PROGRAM F21_ContentHandScanner
VAR
	bDT_HandScanerInUse			: BOOL;
	fbBarcodeType			: FB_SYSTEM_BarcodeType;

	bPackBarcode					: BOOL;
	bOuterIntermediateBarcode		: BOOL;
	bOuterBarcode					: BOOL;
	bCaseBarcode					: BOOL;
	sPackBarcode					: T_PACK_Barcode;
	sOuterIntermediateBarcode		:  T_MaxString;
	sOuterBarcode					: T_OUTER_Barcode;
	sCaseBarcode					: T_CASE_Barcode;

	bLocalCaseBarcode					: BOOL;
	sLocalCaseBarcode					: T_CASE_Barcode;

	fbSearchCaseContent	: FB_SYSTEM_SearchBarcode;

	fbFindOCV_DB			: FB_OCV_FindDB;
	fbFindOAC_DB			: FB_OAC_FindDB;

(*	fbFindOCVFile			: FB_OCV_FindFile;
	stOACData				: ST_OAC_Data;
	sCode				: T_PACK_Barcode;*)

	aOCVRecordDBName		 : ARRAY[1..2] OF T_MaxString;
	sOACRecordName			: T_MaxString;


	fbRestoreCACDataFromDB	:FB_CAC_RestoreDataFromDB;
	sCACFile				: T_MaxString;

	nOCVRestored			: UDINT;
	nOACRestored			: UDINT;
	nCACRestored			: UDINT;

	bOACFound: BOOL;
	bOCVFound: BOOL;
	bOCVValid: BOOL;
	sOuterCodeAI		: T_MaxString;
	(*strPackCodeAI:			STRING(255);*)

	bValidateForOCVDataExistDone :BOOL;
	bValidateForRefeedDone: BOOL;
	bValidateForRefeedOK: BOOL;

	rtrigValidateOCVForDataExistValid			: R_TRIG;
	rtrigValidateOCVForDataExistInvalid			: R_TRIG;
	rtrigValidateOCVForDataNotExist			: R_TRIG;
	tofValidateOCVForDataExisValid			: TOF;
	tofValidateOCVForDataExisInvalid			: TOF;
	tofValidateOCVForDataNotExis				: TOF;


	rtrigValidateOACForRefeedDoneValid		: R_TRIG;
	rtrigValidateOACForRefeedDoneInvalid		: R_TRIG;
	rtrigValidateOACForDataNotExist			: R_TRIG;
	tofValidateOACForRefeedValid			: TOF;
	tofValidateOACForRefeedInvalid			: TOF;
	tofValidateOACForDataNotExis				: TOF;

	rtrigRestoreCACFileDoneValid: R_TRIG;
	rtrigRestoreCACFileDoneInvalid: R_TRIG;
	tofRestoreCACFileValid: TOF;
	tofRestoreCACFileInvalid: TOF;

END_VAR

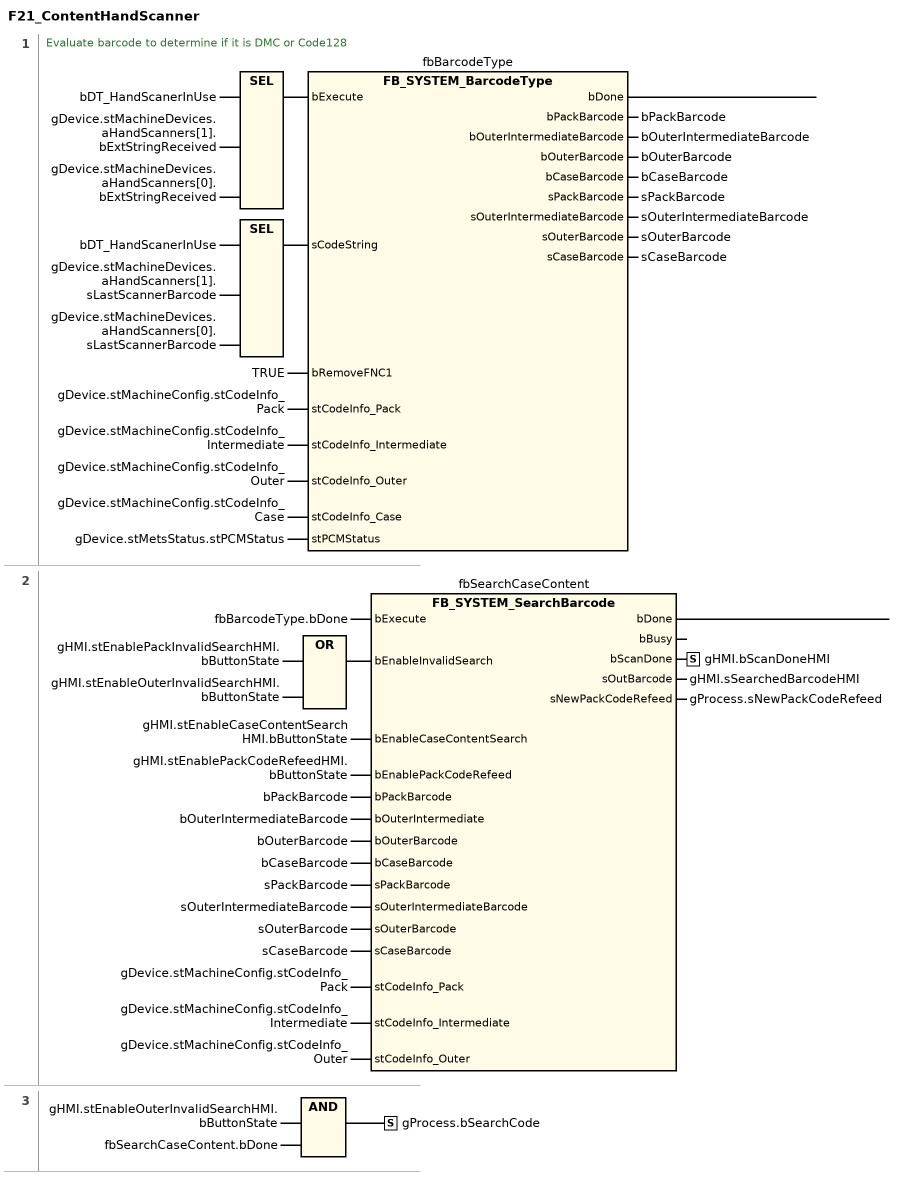
// NETWORK 1
// Evaluate barcode to determine if it is DMC or Code128
fbBarcodeType(
    bExecute := SEL(bDT_HandScanerInUse, gDevice.stMachineDevices.aHandScanners[1].bExtStringReceived, gDevice.stMachineDevices.aHandScanners[0].bExtStringReceived),
    sCodeString := SEL(bDT_HandScanerInUse, gDevice.stMachineDevices.aHandScanners[1].sLastScannerBarcode, gDevice.stMachineDevices.aHandScanners[0].sLastScannerBarcode),
    bRemoveFNC1 := TRUE,
    stCodeInfo_Pack := gDevice.stMachineConfig.stCodeInfo_Pack,
    stCodeInfo_Intermediate := gDevice.stMachineConfig.stCodeInfo_Intermediate,
    stCodeInfo_Outer := gDevice.stMachineConfig.stCodeInfo_Outer,
    stCodeInfo_Case := gDevice.stMachineConfig.stCodeInfo_Case,
    stPCMStatus := gDevice.stMetsStatus.stPCMStatus,
    bPackBarcode => bPackBarcode,
    bOuterIntermediateBarcode => bOuterIntermediateBarcode,
    bOuterBarcode => bOuterBarcode,
    bCaseBarcode => bCaseBarcode,
    sPackBarcode => sPackBarcode,
    sOuterIntermediateBarcode => sOuterIntermediateBarcode,
    sOuterBarcode => sOuterBarcode,
    sCaseBarcode => sCaseBarcode); // FB_SYSTEM_BarcodeType

// NETWORK 2
fbSearchCaseContent(
    bExecute := fbBarcodeType.bDone,
    bEnableInvalidSearch := gHMI.stEnablePackInvalidSearchHMI.bButtonState OR gHMI.stEnableOuterInvalidSearchHMI.bButtonState,
    bEnableCaseContentSearch := gHMI.stEnableCaseContentSearchHMI.bButtonState,
    bEnablePackCodeRefeed := gHMI.stEnablePackCodeRefeedHMI.bButtonState,
    bPackBarcode := bPackBarcode,
    bOuterIntermediate := bOuterIntermediateBarcode,
    bOuterBarcode := bOuterBarcode,
    bCaseBarcode := bCaseBarcode,
    sPackBarcode := sPackBarcode,
    sOuterIntermediateBarcode := sOuterIntermediateBarcode,
    sOuterBarcode := sOuterBarcode,
    sCaseBarcode := sCaseBarcode,
    stCodeInfo_Pack := gDevice.stMachineConfig.stCodeInfo_Pack,
    stCodeInfo_Intermediate := gDevice.stMachineConfig.stCodeInfo_Intermediate,
    stCodeInfo_Outer := gDevice.stMachineConfig.stCodeInfo_Outer,
    sOutBarcode => gHMI.sSearchedBarcodeHMI,
    sNewPackCodeRefeed => gProcess.sNewPackCodeRefeed); // FB_SYSTEM_SearchBarcode
gHMI.bScanDoneHMI S= fbSearchCaseContent.bScanDone;

// NETWORK 3
gProcess.bSearchCode S= gHMI.stEnableOuterInvalidSearchHMI.bButtonState AND fbSearchCaseContent.bDone;

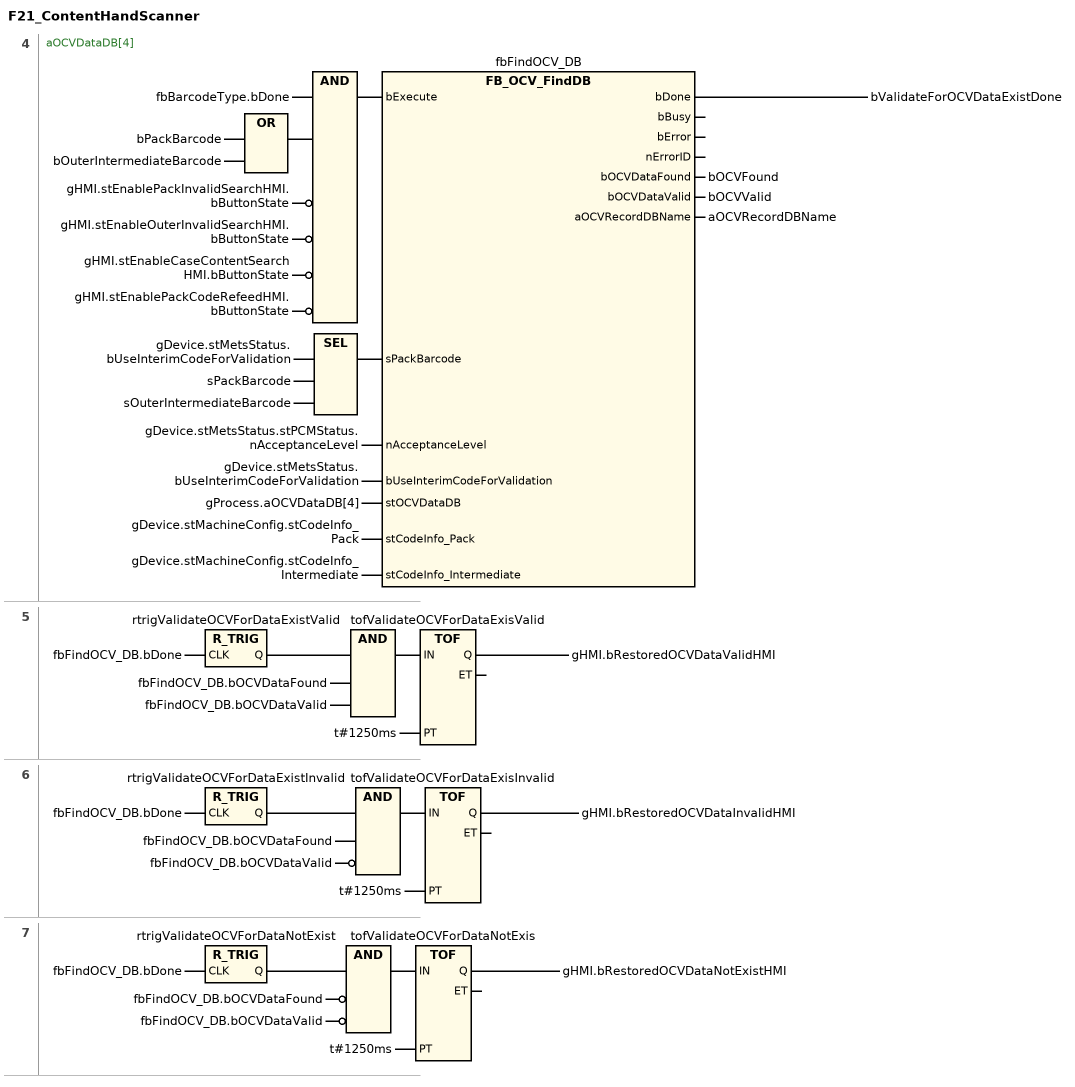
// NETWORK 4
// aOCVDataDB[4]
fbFindOCV_DB(
    bExecute := fbBarcodeType.bDone AND (bPackBarcode OR bOuterIntermediateBarcode) AND NOT gHMI.stEnablePackInvalidSearchHMI.bButtonState AND NOT gHMI.stEnableOuterInvalidSearchHMI.bButtonState AND NOT gHMI.stEnableCaseContentSearchHMI.bButtonState AND NOT gHMI.stEnablePackCodeRefeedHMI.bButtonState,
    sPackBarcode := SEL(gDevice.stMetsStatus.bUseInterimCodeForValidation, sPackBarcode, sOuterIntermediateBarcode),
    nAcceptanceLevel := gDevice.stMetsStatus.stPCMStatus.nAcceptanceLevel,
    bUseInterimCodeForValidation := gDevice.stMetsStatus.bUseInterimCodeForValidation,
    stOCVDataDB := gProcess.aOCVDataDB[4],
    stCodeInfo_Pack := gDevice.stMachineConfig.stCodeInfo_Pack,
    stCodeInfo_Intermediate := gDevice.stMachineConfig.stCodeInfo_Intermediate,
    bOCVDataFound => bOCVFound,
    bOCVDataValid => bOCVValid,
    aOCVRecordDBName => aOCVRecordDBName); // FB_OCV_FindDB
bValidateForOCVDataExistDone := fbFindOCV_DB.bDone;

// NETWORK 5
rtrigValidateOCVForDataExistValid(CLK := fbFindOCV_DB.bDone); // R_TRIG
tofValidateOCVForDataExisValid(IN := rtrigValidateOCVForDataExistValid.Q AND fbFindOCV_DB.bOCVDataFound AND fbFindOCV_DB.bOCVDataValid, PT := t#1250ms); // TOF
gHMI.bRestoredOCVDataValidHMI := tofValidateOCVForDataExisValid.Q;

// NETWORK 6
rtrigValidateOCVForDataExistInvalid(CLK := fbFindOCV_DB.bDone); // R_TRIG
tofValidateOCVForDataExisInvalid(IN := rtrigValidateOCVForDataExistInvalid.Q AND fbFindOCV_DB.bOCVDataFound AND NOT fbFindOCV_DB.bOCVDataValid, PT := t#1250ms); // TOF
gHMI.bRestoredOCVDataInvalidHMI := tofValidateOCVForDataExisInvalid.Q;

// NETWORK 7
rtrigValidateOCVForDataNotExist(CLK := fbFindOCV_DB.bDone); // R_TRIG
tofValidateOCVForDataNotExis(IN := rtrigValidateOCVForDataNotExist.Q AND NOT fbFindOCV_DB.bOCVDataFound AND NOT fbFindOCV_DB.bOCVDataValid, PT := t#1250ms); // TOF
gHMI.bRestoredOCVDataNotExistHMI := tofValidateOCVForDataNotExis.Q;

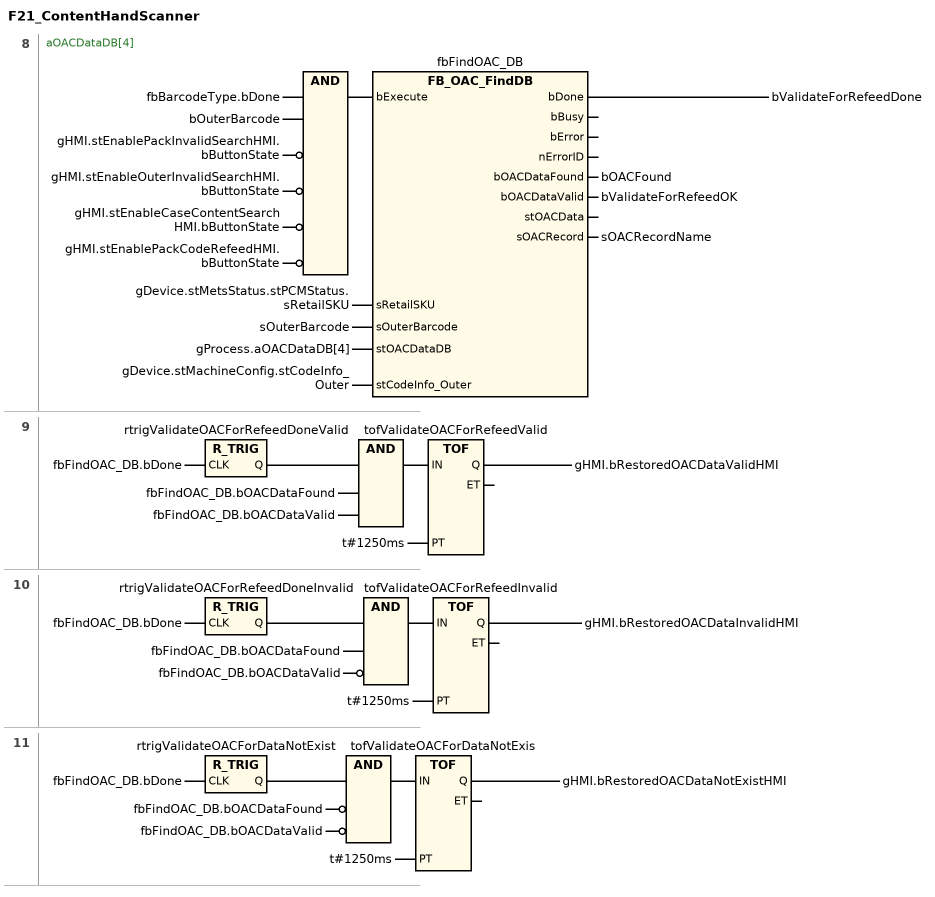
// NETWORK 8
// aOACDataDB[4]
fbFindOAC_DB(
    bExecute := fbBarcodeType.bDone AND bOuterBarcode AND NOT gHMI.stEnablePackInvalidSearchHMI.bButtonState AND NOT gHMI.stEnableOuterInvalidSearchHMI.bButtonState AND NOT gHMI.stEnableCaseContentSearchHMI.bButtonState AND NOT gHMI.stEnablePackCodeRefeedHMI.bButtonState,
    sRetailSKU := gDevice.stMetsStatus.stPCMStatus.sRetailSKU,
    sOuterBarcode := sOuterBarcode,
    stOACDataDB := gProcess.aOACDataDB[4],
    stCodeInfo_Outer := gDevice.stMachineConfig.stCodeInfo_Outer,
    bOACDataFound => bOACFound,
    bOACDataValid => bValidateForRefeedOK,
    sOACRecord => sOACRecordName); // FB_OAC_FindDB
bValidateForRefeedDone := fbFindOAC_DB.bDone;

// NETWORK 9
rtrigValidateOACForRefeedDoneValid(CLK := fbFindOAC_DB.bDone); // R_TRIG
tofValidateOACForRefeedValid(IN := rtrigValidateOACForRefeedDoneValid.Q AND fbFindOAC_DB.bOACDataFound AND fbFindOAC_DB.bOACDataValid, PT := t#1250ms); // TOF
gHMI.bRestoredOACDataValidHMI := tofValidateOACForRefeedValid.Q;

// NETWORK 10
rtrigValidateOACForRefeedDoneInvalid(CLK := fbFindOAC_DB.bDone); // R_TRIG
tofValidateOACForRefeedInvalid(IN := rtrigValidateOACForRefeedDoneInvalid.Q AND fbFindOAC_DB.bOACDataFound AND NOT fbFindOAC_DB.bOACDataValid, PT := t#1250ms); // TOF
gHMI.bRestoredOACDataInvalidHMI := tofValidateOACForRefeedInvalid.Q;

// NETWORK 11
rtrigValidateOACForDataNotExist(CLK := fbFindOAC_DB.bDone); // R_TRIG
tofValidateOACForDataNotExis(IN := rtrigValidateOACForDataNotExist.Q AND NOT fbFindOAC_DB.bOACDataFound AND NOT fbFindOAC_DB.bOACDataValid, PT := t#1250ms); // TOF
gHMI.bRestoredOACDataNotExistHMI := tofValidateOACForDataNotExis.Q;

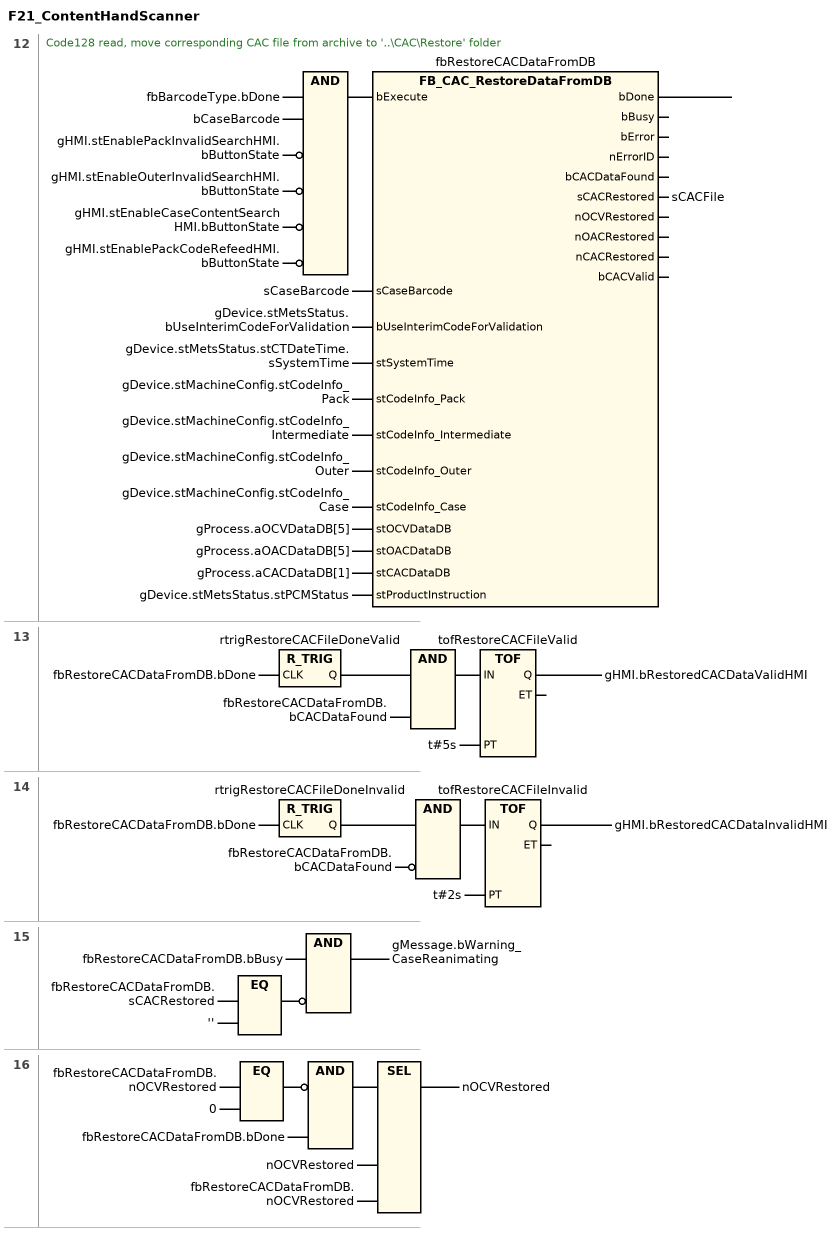
// NETWORK 12
// Code128 read, move corresponding CAC file from archive to '..\CAC\Restore' folder
fbRestoreCACDataFromDB(
    bExecute := fbBarcodeType.bDone AND bCaseBarcode AND NOT gHMI.stEnablePackInvalidSearchHMI.bButtonState AND NOT gHMI.stEnableOuterInvalidSearchHMI.bButtonState AND NOT gHMI.stEnableCaseContentSearchHMI.bButtonState AND NOT gHMI.stEnablePackCodeRefeedHMI.bButtonState,
    sCaseBarcode := sCaseBarcode,
    bUseInterimCodeForValidation := gDevice.stMetsStatus.bUseInterimCodeForValidation,
    stSystemTime := gDevice.stMetsStatus.stCTDateTime.sSystemTime,
    stCodeInfo_Pack := gDevice.stMachineConfig.stCodeInfo_Pack,
    stCodeInfo_Intermediate := gDevice.stMachineConfig.stCodeInfo_Intermediate,
    stCodeInfo_Outer := gDevice.stMachineConfig.stCodeInfo_Outer,
    stCodeInfo_Case := gDevice.stMachineConfig.stCodeInfo_Case,
    stOCVDataDB := gProcess.aOCVDataDB[5],
    stOACDataDB := gProcess.aOACDataDB[5],
    stCACDataDB := gProcess.aCACDataDB[1],
    stProductInstruction := gDevice.stMetsStatus.stPCMStatus,
    sCACRestored => sCACFile); // FB_CAC_RestoreDataFromDB

// NETWORK 13
rtrigRestoreCACFileDoneValid(CLK := fbRestoreCACDataFromDB.bDone); // R_TRIG
tofRestoreCACFileValid(IN := rtrigRestoreCACFileDoneValid.Q AND fbRestoreCACDataFromDB.bCACDataFound, PT := t#5s); // TOF
gHMI.bRestoredCACDataValidHMI := tofRestoreCACFileValid.Q;

// NETWORK 14
rtrigRestoreCACFileDoneInvalid(CLK := fbRestoreCACDataFromDB.bDone); // R_TRIG
tofRestoreCACFileInvalid(IN := rtrigRestoreCACFileDoneInvalid.Q AND NOT fbRestoreCACDataFromDB.bCACDataFound, PT := t#2s); // TOF
gHMI.bRestoredCACDataInvalidHMI := tofRestoreCACFileInvalid.Q;

// NETWORK 15
gMessage.bWarning_CaseReanimating := fbRestoreCACDataFromDB.bBusy AND NOT (fbRestoreCACDataFromDB.sCACRestored = '');

// NETWORK 16
nOCVRestored := SEL(NOT (fbRestoreCACDataFromDB.nOCVRestored = 0) AND fbRestoreCACDataFromDB.bDone, nOCVRestored, fbRestoreCACDataFromDB.nOCVRestored);

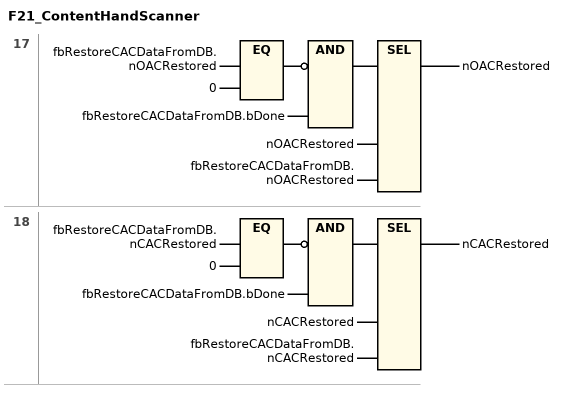
// NETWORK 17
nOACRestored := SEL(NOT (fbRestoreCACDataFromDB.nOACRestored = 0) AND fbRestoreCACDataFromDB.bDone, nOACRestored, fbRestoreCACDataFromDB.nOACRestored);

// NETWORK 18
nCACRestored := SEL(NOT (fbRestoreCACDataFromDB.nCACRestored = 0) AND fbRestoreCACDataFromDB.bDone, nCACRestored, fbRestoreCACDataFromDB.nCACRestored);

END_PROGRAM

(* stored: Version 1.1.0.1
   POU F21_ContentHandScanner: Id {d063a5fb-23d7-4aa2-8757-789d92c1a4d3}, SpecialFunc None *)
